TYPE
    ST_FanucRobotList :
    STRUCT
        StorageRobot  : FB_FanucRobot_Basic;
        ShippingRobot : FB_FanucRobot_Basic;
    END_STRUCT
END_TYPE

(* stored: Version 1.1.0.1, ProductVersion 3.1.4024.13
   DUT ST_FanucRobotList: Id {d88d2db0-da63-4f1f-997f-d6be6a2b963d} *)
